Staubli VAL3: stringToJoints.pgx

program stringToJoints(string x_sStr (dimensions=1), joint& x_jTemp[] (dimensions=1))
  local string l_sX
  local string l_sY
  local num l_nPosX
  local num l_nPosY
  local bool l_bOk
  local num l_nPosZ
  local string l_sZ
  local bool l_bTemp
  local num l_ni
  local string l_sRX
  local string l_sRY
  local string l_sRZ
  local num l_nPosRX
  local num l_nPosRY
  local num l_nPosRZ
  local num l_nDbg
  local point l_ptest
begin
  //  l_sX=mid(x_sStr,7,13)
  //  call FC_chrdeal(l_sX)
  //  l_sY=mid(x_sStr,7,23)
  //  call FC_chrdeal(l_sY)
  //  l_sZ=mid(x_sStr,7,33)
  //  call FC_chrdeal(l_sZ)
  //  l_sRX=mid(x_sStr,7,43)
  //  call FC_chrdeal(l_sRX)
  //  l_sRY=mid(x_sStr,7,53)
  //  call FC_chrdeal(l_sRY)
  //  l_sRZ=mid(x_sStr,7,63)
  //  call FC_chrdeal(l_sRZ)
  //  toNum(l_sX,l_nPosX,l_bOk)
  //  toNum(l_sY,l_nPosY,l_bOk)
  //  toNum(l_sZ,l_nPosZ,l_bOk)
  //  toNum(l_sRX,l_nPosRX,l_bOk)
  //  toNum(l_sRY,l_nPosRY,l_bOk)
  //  toNum(l_sRZ,l_nPosRZ,l_bOk)
  //
  //  MoveTo.trsf.x=l_nPosX
  //  MoveTo.trsf.y=l_nPosY
  //  MoveTo.trsf.z=l_nPosZ
  //  MoveTo.trsf.rx=l_nPosRX
  //  MoveTo.trsf.ry=l_nPosRY
  //  MoveTo.trsf.rz=l_nPosRZ
  //  //MoveTo=position(l_ptest,FrmDraw)
  //  l_bTemp=pointToJoint(tTool,jConfig,MoveTo,x_jTemp)
  //  if l_bTemp==false
  //    io:socket="(RBERRO)"
  //    popUpMsg("wrong point position!!!")
  //  endIf
end
